// TIA Portal V20 export
TYPE "IO_Device_Functinal_Test"
   STRUCT
      Life_Trigger_PLC_Functional_Test_2 : Bool;
      Star_Test_PLC_Functional_Test_2 : Bool;
      Button_PLC_Functional_Test_2 : Bool;
      Electrical_Current_Test_Approved_PLC_Functional_Test_2 : Bool;
      Visual_Test_Approved_PLC_Functional_Test_2 : Bool;
      Electrical_Current_Read_PLC_Functional_Test_2 : UInt;
      Life_Trigger_PLC_Functional_Test_4 : Bool;
      Star_Test_PLC_Functional_Test_4 : Bool;
      Button_PLC_Functional_Test_4 : Bool;
      Electrical_Current_Test_Approved_PLC_Functional_Test_4 : Bool;
      Visual_Test_Approved_PLC_Functional_Test_4 : Bool;
      Electrical_Current_Read_PLC_Functional_Test_4 : UInt;
      Life_Trigger_PLC_Functional_Test_6 : Bool;
      Star_Test_PLC_Functional_Test_6 : Bool;
      Button_PLC_Functional_Test_6 : Bool;
      Electrical_Current_Test_Approved_PLC_Functional_Test_6 : Bool;
      Visual_Test_Approved_PLC_Functional_Test_6 : Bool;
      Electrical_Current_Read_PLC_Functional_Test_6 : UInt;
      Life_Trigger_PLC_Functional_Test_8 : Bool;
      Star_Test_PLC_Functional_Test_8 : Bool;
      Button_PLC_Functional_Test_8 : Bool;
      Electrical_Current_Test_Approved_PLC_Functional_Test_8 : Bool;
      Visual_Test_Approved_PLC_Functional_Test_8 : Bool;
      Electrical_Current_Read_PLC_Functional_Test_8 : UInt;
      Life_Trigger_PLC_Functional_Test_10 : Bool;
      Star_Test_PLC_Functional_Test_10 : Bool;
      Button_PLC_Functional_Test_10 : Bool;
      Electrical_Current_Test_Approved_PLC_Functional_Test_10 : Bool;
      Visual_Test_Approved_PLC_Functional_Test_10 : Bool;
      Electrical_Current_Read_PLC_Functional_Test_10 : UInt;
      Life_Trigger_PLC_Functional_Test_12 : Bool;
      Star_Test_PLC_Functional_Test_12 : Bool;
      Button_PLC_Functional_Test_12 : Bool;
      Electrical_Current_Test_Approved_PLC_Functional_Test_12 : Bool;
      Visual_Test_Approved_PLC_Functional_Test_12 : Bool;
      Electrical_Current_Read_PLC_Functional_Test_12 : UInt;
      Life_Trigger_PLC_Functional_Test_14 : Bool;
      Star_Test_PLC_Functional_Test_14 : Bool;
      Button_PLC_Functional_Test_14 : Bool;
      Electrical_Current_Test_Approved_PLC_Functional_Test_14 : Bool;
      Visual_Test_Approved_PLC_Functional_Test_14 : Bool;
      Electrical_Current_Read_PLC_Functional_Test_14 : UInt;
      Life_Trigger_PLC_Functional_Test_16 : Bool;
      Star_Test_PLC_Functional_Test_16 : Bool;
      Button_PLC_Functional_Test_16 : Bool;
      Electrical_Current_Test_Approved_PLC_Functional_Test_16 : Bool;
      Visual_Test_Approved_PLC_Functional_Test_16 : Bool;
      Electrical_Current_Read_PLC_Functional_Test_16 : UInt;
      Life_Trigger_PLC_Functional_Test_18 : Bool;
      Star_Test_PLC_Functional_Test_18 : Bool;
      Button_PLC_Functional_Test_18 : Bool;
      Electrical_Current_Test_Approved_PLC_Functional_Test_18 : Bool;
      Visual_Test_Approved_PLC_Functional_Test_18 : Bool;
      Electrical_Current_Read_PLC_Functional_Test_18 : UInt;
      Life_Trigger_PLC_Functional_Test_20 : Bool;
      Star_Test_PLC_Functional_Test_20 : Bool;
      Button_PLC_Functional_Test_20 : Bool;
      Electrical_Current_Test_Approved_PLC_Functional_Test_20 : Bool;
      Visual_Test_Approved_PLC_Functional_Test_20 : Bool;
      Electrical_Current_Read_PLC_Functional_Test_20 : UInt;
      Life_Trigger_PLC_Functional_Test_22 : Bool;
      Star_Test_PLC_Functional_Test_22 : Bool;
      Button_PLC_Functional_Test_22 : Bool;
      Electrical_Current_Test_Approved_PLC_Functional_Test_22 : Bool;
      Visual_Test_Approved_PLC_Functional_Test_22 : Bool;
      Electrical_Current_Read_PLC_Functional_Test_22 : UInt;
      Life_Trigger_PLC_Functional_Test_24 : Bool;
      Star_Test_PLC_Functional_Test_24 : Bool;
      Button_PLC_Functional_Test_24 : Bool;
      Electrical_Current_Test_Approved_PLC_Functional_Test_24 : Bool;
      Visual_Test_Approved_PLC_Functional_Test_24 : Bool;
      Electrical_Current_Read_PLC_Functional_Test_24 : UInt;
      Life_Trigger_PLC_Functional_Test_26 : Bool;
      Star_Test_PLC_Functional_Test_26 : Bool;
      Button_PLC_Functional_Test_26 : Bool;
      Electrical_Current_Test_Approved_PLC_Functional_Test_26 : Bool;
      Visual_Test_Approved_PLC_Functional_Test_26 : Bool;
      Electrical_Current_Read_PLC_Functional_Test_26 : UInt;
      Life_Trigger_PLC_Functional_Test_28 : Bool;
      Star_Test_PLC_Functional_Test_28 : Bool;
      Button_PLC_Functional_Test_28 : Bool;
      Electrical_Current_Test_Approved_PLC_Functional_Test_28 : Bool;
      Visual_Test_Approved_PLC_Functional_Test_28 : Bool;
      Electrical_Current_Read_PLC_Functional_Test_28 : UInt;
      Life_Trigger_PLC_Functional_Test_30 : Bool;
      Star_Test_PLC_Functional_Test_30 : Bool;
      Button_PLC_Functional_Test_30 : Bool;
      Electrical_Current_Test_Approved_PLC_Functional_Test_30 : Bool;
      Visual_Test_Approved_PLC_Functional_Test_30 : Bool;
      Electrical_Current_Read_PLC_Functional_Test_30 : UInt;
   END_STRUCT;
END_TYPE
